RoboDK station: experimentation_nachiket.rdk

Station experimentation_nachiket (saved by RoboDK 5.2.3). Poses are relative to the parent item; angles as X-Y-Z fixed-axis rotations.
